// TIA Portal project "MobileLLRF" (V18)

(* hardware
DEVICE "S7-1200 station_1"  S7-1200 Station
   slot 0: "Rack_0"  S7-1200 Rack  Rack  V1.0
   slot 1: "PLC_1"  CPU 1212C DC/DC/DC  6ES7 212-1AE40-0XB0  V4.6
   slot 3: "AQ 1x12BIT_1"  AQ1 signal board  6ES7 232-4HA30-0XB0  V1.0
*)

// ===== PLC "PLC_1"  CPU 1212C DC/DC/DC =====

VAR_GLOBAL   // PLC tag table "Default tag table"
   "System_Byte" AT %MB1 : Byte;
   "FirstScan" AT %M1.0 : Bool;
   "DiagStatusUpdate" AT %M1.1 : Bool;
   "AlwaysTRUE" AT %M1.2 : Bool;
   "AlwaysFALSE" AT %M1.3 : Bool;
   "Clock_Byte" AT %MB0 : Byte;
   "Clock_10Hz" AT %M0.0 : Bool;
   "Clock_5Hz" AT %M0.1 : Bool;
   "Clock_2.5Hz" AT %M0.2 : Bool;
   "Clock_2Hz" AT %M0.3 : Bool;
   "Clock_1.25Hz" AT %M0.4 : Bool;
   "Clock_1Hz" AT %M0.5 : Bool;
   "Clock_0.625Hz" AT %M0.6 : Bool;
   "Clock_0.5Hz" AT %M0.7 : Bool;
END_VAR

VAR_GLOBAL   // PLC tag table "In/Out"
   "DigitalInputs" AT %IB0 : Byte;
   "DigitalOutputs" AT %QB0 : Byte;
   "AI0" AT %IW64 : Int;
   "AI1" AT %IW66 : Int;
   "TestDO" AT %Q0.5 : Bool;
   "AQ0" AT %QW80 : Int;
   "AI_Combined" AT %ID64 : DWord;
   "TriggerLED" AT %Q0.0 : Bool;
END_VAR

TYPE "PLC2Epics_TYPE"
   STRUCT
      CavPos0 : Bool;
      CavPos1 : Bool;
      CavPos2 : Bool;
      RFswitchON : Bool;
      StepAtten10dB : Bool;
      StepAtten20dB : Bool;
      StepAtten40dB : Bool;
      SSPAenabled : Bool;
      ExtIntrlk : Bool;
      VCA_Ctrl : Real;
      spare : Array[0..9] of Word;
   END_STRUCT;
END_TYPE

TYPE "Epics2PLC_TYPE"
   STRUCT
      StepAtten10dB : Bool;
      StepAtten20dB : Bool;
      StepAtten40dB : Bool;
      RFswitchON : Bool;
      EnableSSPA : Bool;
      VCA_Ctrl : Real;
      spare : Array[0..9] of Word;
   END_STRUCT;
END_TYPE

TYPE "CommParam"
VERSION : 0.1
   STRUCT
      interface_id : Word;   // HW-identifier of IE-interface submodule
      conn_id : Word;   // Connection reference / identifier
      connection_type : Byte := 16#000B;   // Type of connection: 11=TCP/IP, 19=UDP (17=TCP/IP) ??B#16#11??
      active_established : Bool := False;   // active/passive connection establishment
      local_port : UInt;   // local UDP/TCP port number
      init_com : Bool;   // send_db : INT; recv_db : INT;
      send_len : UDInt;
      recv_len : UDInt;
      sendtrigger : Bool;
      sendtime : Time_Of_Day;
      sendinterval : DInt;
   END_STRUCT;
END_TYPE

// folder: EPICS_Communication

DATA_BLOCK "CH_PARAM_TCP"   // DB300
{ S7_Optimized_Access := 'FALSE' }
VERSION : 0.1
   VAR
      CommParam : "CommParam";
   END_VAR
BEGIN
   CommParam.send_len := 26;
   CommParam.recv_len := 26;
   CommParam.sendinterval := DINT#500;
   CommParam.local_port := 3000;
   CommParam.interface_id := 64;
   CommParam.conn_id := 3;
   CommParam.connection_type := 16#000b;
END_DATA_BLOCK

DATA_BLOCK "TCP1_instance"   // DB310
{ S7_Optimized_Access := 'FALSE' }
AUTHOR : CSL
FAMILY : TSTMP
NAME : S_R_TCP1
VERSION : 1.0
// stored: InstanceOfName Tsend_Trecv
"Tsend_Trecv"
BEGIN
END_DATA_BLOCK

// folder: Epics

DATA_BLOCK "PLC2Epics"   // DB100
{ S7_Optimized_Access := 'FALSE' }
VERSION : 0.1
   VAR
      DATA : "PLC2Epics_TYPE";
   END_VAR
BEGIN
END_DATA_BLOCK

DATA_BLOCK "Epics2PLC"   // DB101
{ S7_Optimized_Access := 'FALSE' }
VERSION : 0.1
   VAR
      data : "Epics2PLC_TYPE";
   END_VAR
BEGIN
END_DATA_BLOCK

// folder: Input/Output

DATA_BLOCK "#ANALOG_IN"   // DB400
{ S7_Optimized_Access := 'FALSE' }
VERSION : 0.1
   VAR
      Spare1 : Int;
      Spare2 : Int;
   END_VAR
BEGIN
END_DATA_BLOCK

DATA_BLOCK "#ANALOG_OUT"   // DB401
{ S7_Optimized_Access := 'FALSE' }
VERSION : 0.1
   VAR
      VCA_Ctrl : Word;
   END_VAR
BEGIN
END_DATA_BLOCK

DATA_BLOCK "#DIGITAL_INPUTS"   // DB402
{ S7_Optimized_Access := 'FALSE' }
VERSION : 0.1
   VAR
      CavPos0 : Bool;   // Coded LLRF connection to DUT (LSB)
      CavPos1 : Bool;   // Coded LLRF connection to DUT
      CavPos2 : Bool;   // Coded LLRF connection to DUT (MSB)
      RFswitchOn : Bool;
      ExtIntlk : Bool;
      Spare2 : Bool;
      Spare3 : Bool;
      Spare4 : Bool;
   END_VAR
BEGIN
END_DATA_BLOCK

DATA_BLOCK "#DIGITAL_OUTPUTS"   // DB403
{ S7_Optimized_Access := 'FALSE' }
VERSION : 0.1
   VAR
      StepAtt10dB : Bool;
      StepAtt20dB : Bool;
      StepAtt40dB : Bool;
      RFswitchOff : Bool;
      RFswitchOn : Bool;
      EnableSSPA : Bool;
   END_VAR
BEGIN
END_DATA_BLOCK

// folder: (top level)

FUNCTION "Process" : Void   // FC103, LAD
TITLE = Process logic
{ S7_Optimized_Access := 'TRUE' }
VERSION : 0.1
BEGIN

REGION Network 1
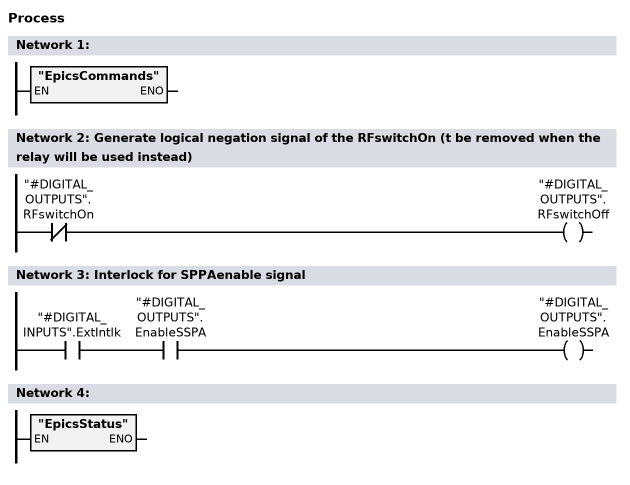
   RUNG wire#powerrail
      "EpicsCommands"()
   END_RUNG
   // the same network as SCL:
   "EpicsCommands"();
END_REGION

REGION Network 2: Generate logical negation signal of the RFswitchOn (t be removed when the relay will be used instead)
   RUNG wire#powerrail
      I_Contact( "#DIGITAL_OUTPUTS".RFswitchOn )
      Coil( "#DIGITAL_OUTPUTS".RFswitchOff )
   END_RUNG
   // the same network as SCL:
   "#DIGITAL_OUTPUTS".RFswitchOff := NOT "#DIGITAL_OUTPUTS".RFswitchOn;
END_REGION

REGION Network 3: Interlock for SPPAenable signal
   RUNG wire#powerrail
      Contact( "#DIGITAL_INPUTS".ExtIntlk )
      Contact( "#DIGITAL_OUTPUTS".EnableSSPA )
      Coil( "#DIGITAL_OUTPUTS".EnableSSPA )
   END_RUNG
   // the same network as SCL:
   "#DIGITAL_OUTPUTS".EnableSSPA := "#DIGITAL_INPUTS".ExtIntlk AND "#DIGITAL_OUTPUTS".EnableSSPA;
END_REGION

REGION Network 4
   RUNG wire#powerrail
      "EpicsStatus"()
   END_RUNG
   // the same network as SCL:
   "EpicsStatus"();
END_REGION
END_FUNCTION

ORGANIZATION_BLOCK "Main"   // OB1, LAD, ProgramCycle
TITLE = "Main Program Sweep (Cycle)"
{ S7_Optimized_Access := 'TRUE' }
VERSION : 0.1
   VAR_INPUT
      Initial_Call : Bool;   // Initial call of this OB
      Remanence : Bool;   // =True, if remanent data are available
   END_VAR
BEGIN

REGION Network 1
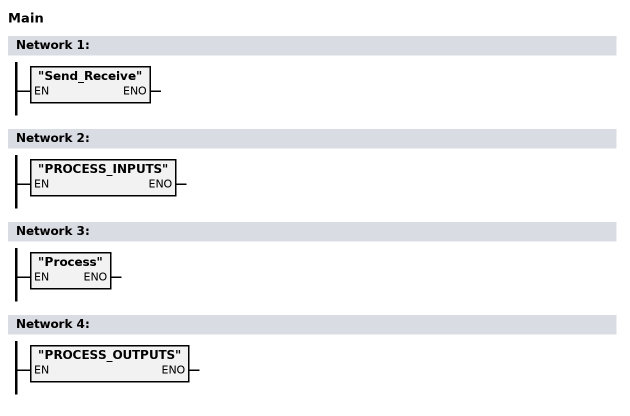
   RUNG wire#powerrail
      "Send_Receive"()
   END_RUNG
   // the same network as SCL:
   "Send_Receive"();
END_REGION

REGION Network 2
   RUNG wire#powerrail
      "PROCESS_INPUTS"()
   END_RUNG
   // the same network as SCL:
   "PROCESS_INPUTS"();
END_REGION

REGION Network 3
   RUNG wire#powerrail
      "Process"()
   END_RUNG
   // the same network as SCL:
   "Process"();
END_REGION

REGION Network 4
   RUNG wire#powerrail
      "PROCESS_OUTPUTS"()
   END_RUNG
   // the same network as SCL:
   "PROCESS_OUTPUTS"();
END_REGION
END_ORGANIZATION_BLOCK

ORGANIZATION_BLOCK "Startup"   // OB100, LAD, Startup
TITLE = "Complete Restart"
{ S7_Optimized_Access := 'TRUE' }
VERSION : 0.1
   VAR_INPUT
      LostRetentive : Bool;   // True if retentive data are lost
      LostRTC : Bool;   // True if date and time are lost
   END_VAR
BEGIN

REGION Network 1
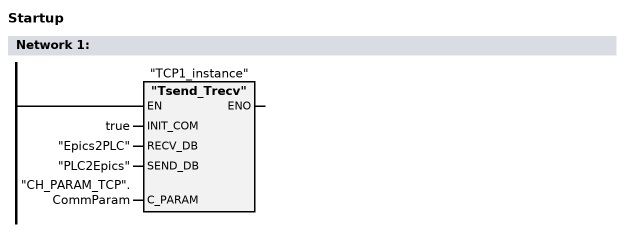
   RUNG wire#powerrail
      "TCP1_instance"(INIT_COM := true, RECV_DB := "Epics2PLC", SEND_DB := "PLC2Epics", C_PARAM := "CH_PARAM_TCP".CommParam)
   END_RUNG
   // the same network as SCL:
   "TCP1_instance"(INIT_COM := true,   // "Tsend_Trecv"
                   RECV_DB := "Epics2PLC",
                   SEND_DB := "PLC2Epics",
                   C_PARAM := "CH_PARAM_TCP".CommParam);
END_REGION
END_ORGANIZATION_BLOCK

// folder: EPICS_Communication

FUNCTION_BLOCK "Tsend_Trecv"   // FB300, SCL
TITLE = TCP1 send receive channel
{ S7_Optimized_Access := 'FALSE' }
AUTHOR : CSL
FAMILY : TSTMP
NAME : S_R_TCP1
VERSION : 1.0
   VAR_INPUT
      INIT_COM : Bool;
      RECV_DB : Variant;
      SEND_DB : Variant;
   END_VAR
   VAR_IN_OUT
      C_PARAM : "CommParam";
   END_VAR
   VAR
      T_SEND : TSEND;
      T_RECV : TRCV;
      T_CONN : TCON;
      T_PARAM : TCON_IP_v4;
      COM1 : Struct
         CONNECTED : Bool;
         CONN_DONE : Bool;
         CONN_BUSY : Bool;
         CONN_ERROR : Bool;
         CONN_STATUS : Word;
         CONN_SETA : Bool;
         SEND_REQ : Bool;
         SEND_DONE : Bool;
         SEND_BUSY : Bool;
         SEND_ERROR : Bool;
         SEND_REQ_P : Bool;
         SEND_STATUS : Word;
         ACT_SEND : Bool;
         RECV_NDR : Bool;
         RECV_BUSY : Bool;
         RECV_ERROR : Bool;
         RECV_STATUS : Word;
         RECV_LEN : UDInt;
      END_STRUCT;
      PLC_COUNT : UDInt;
      CURRENT_DT : DTL;
   END_VAR
   VAR_TEMP
      current_time : Time;
      TIME_DIFF : DInt;
      SEND_TIME : DInt;
      stat : Int;
      tod : Time_Of_Day;
   END_VAR
   VAR CONSTANT
      DAY_IN_MS : DInt := 86400000;
   END_VAR
BEGIN

   // Set communication initialisation bit at restart
   #C_PARAM.init_com := #INIT_COM;

   //Clear Bits to start initial connection and communication
   IF #C_PARAM.init_com THEN
       #COM1.CONNECTED := FALSE;
       #COM1.SEND_REQ := FALSE;
       #COM1.CONN_SETA := FALSE;
   END_IF;

   //set TCPx connection parametres 
   #T_PARAM.InterfaceId :=  WORD_TO_UINT (#C_PARAM.interface_id);
   #T_PARAM.ID := #C_PARAM.conn_id;
   #T_PARAM.ConnectionType := #C_PARAM.connection_type;
   #T_PARAM.ActiveEstablished := #C_PARAM.active_established;
   //T_PARAM.RemotePort := 0; 
   #T_PARAM.LocalPort := #C_PARAM.local_port;

   //Establish TCP connection
   //After the connection has been established, it is automatically monitored and maintained by the operating system of the CPU.
   //If the connection has been interrupted, by any line break or due to the remote communications partner, the active partner attempts to reestablish the connection.
   //Therefore, the FB 65 "TCON" may not be called again! 
   IF NOT #COM1.CONNECTED THEN
       #T_CONN(REQ := #COM1.CONN_SETA,
               ID := #C_PARAM.conn_id,
               DONE => #COM1.CONN_DONE,
               BUSY => #COM1.CONN_BUSY,
               ERROR => #COM1.CONN_ERROR,
               STATUS => #COM1.CONN_STATUS,
               CONNECT := #T_PARAM);
   END_IF;

   //Establish connection
   //While startup phase (initial).
   //Indication of the connection status:
   //a) If the CPU may establish the specified connection after Stop/Run immediately, the variable "CONNECTED" indicates HIGH (=1).
   //b) If the CPU is not able to establish the specified connection after Stop/Run, the variable "CONNECTED" remains LOW(=0).
   //c) Note: If the instance DB is loaded by the user, the variable "CONNECTED" indicates HIGH, although the connection may not be established yet. 
   //However, the FB64 "TRCV" would indicate the STATUS=0x80C4, as long as the connection has NOT been established. 
   IF #C_PARAM.init_com THEN
       #COM1.CONN_SETA := TRUE;
   END_IF;
   IF #COM1.CONN_DONE THEN
       #COM1.CONN_SETA := FALSE;
       #C_PARAM.init_com := FALSE;
   END_IF;
   IF #COM1.CONN_SETA THEN
       #COM1.CONNECTED := FALSE;
   ELSE
       #COM1.CONNECTED := TRUE;
   END_IF;

   //generate send trigger pulse
   //#current_time := TIME_TCK(); // Not available in S/-1200 
   #stat := RD_SYS_T(#CURRENT_DT); // TIME & DATE
   #tod := DTL_TO_TOD(#CURRENT_DT); // Time of Day (ms after midnight)
   #TIME_DIFF := TOD_TO_DINT(#tod) - TOD_TO_DINT(#C_PARAM.sendtime);
   IF (#TIME_DIFF < 0) THEN
       #TIME_DIFF := #TIME_DIFF + #DAY_IN_MS;
   END_IF;
   IF (#C_PARAM.sendinterval < #TIME_DIFF + 1) THEN
       #C_PARAM.sendtrigger := TRUE;
       #SEND_TIME := TOD_TO_DINT(#C_PARAM.sendtime) + #C_PARAM.sendinterval;
       IF (#SEND_TIME >= #DAY_IN_MS) THEN
           #SEND_TIME := #SEND_TIME - #DAY_IN_MS;
       END_IF;
       #C_PARAM.sendtime := DINT_TO_TOD(#SEND_TIME);
       #COM1.SEND_REQ_P := FALSE;
   END_IF;
   //IF (#C_PARAM.sendinterval < ABS(TIME_TO_DINT(#current_time - #C_PARAM.sendtime)) + 1) THEN
   //    #C_PARAM.sendtrigger := TRUE;
   //    #C_PARAM.sendtime := #C_PARAM.sendtime + DINT_TO_TIME(#C_PARAM.sendinterval);  //#C_PARAM.sendtime := #current_time;
   //    #COM1.SEND_REQ_P := FALSE;
   // END_IF;

   //Invoke T_SEND function. 
   //IF connection is established TO transmit the data TO the partner as a message.
   // DATA and LEN from input C_PARAM
   IF #COM1.CONNECTED THEN
       #T_SEND(REQ := #COM1.SEND_REQ,
               ID := #C_PARAM.conn_id,
               LEN := #C_PARAM.send_len,
               DONE => #COM1.SEND_DONE,
               BUSY => #COM1.SEND_BUSY,
               ERROR => #COM1.SEND_ERROR,
               STATUS => #COM1.SEND_STATUS,
               DATA := #SEND_DB);//"datatoIOC_TCP1".CommToIOC);
   END_IF;

   //Generate the rising edge SEND_REQ to start the T_SEND function. 
   IF #C_PARAM.sendtrigger AND NOT #COM1.SEND_REQ_P AND NOT #COM1.SEND_BUSY THEN
        #COM1.SEND_REQ := TRUE;
   END_IF;
   #COM1.SEND_REQ_P := #C_PARAM.sendtrigger;

   IF #COM1.SEND_DONE OR #COM1.SEND_ERROR THEN
       #COM1.SEND_REQ := FALSE;
       #C_PARAM.sendtrigger := FALSE;
   END_IF;


   //Invoke T_RECV function
   //The data is stored into the buffer specified with DATA parameter. 
   //After the data has been received, the data is immediately available in the receive buffer. 
   //Receiving is indicated BY the NDR output parameter.
   //Note: DATA and LEN from input C_PARAM 
   IF #COM1.CONNECTED THEN
       #T_RECV(EN_R := #COM1.CONNECTED,
               ID := #C_PARAM.conn_id,
               LEN := #C_PARAM.recv_len,
               ADHOC := false,
               NDR => #COM1.RECV_NDR,
               BUSY => #COM1.RECV_BUSY,
               ERROR => #COM1.RECV_ERROR,
               STATUS => #COM1.RECV_STATUS,
               RCVD_LEN => #COM1.RECV_LEN,
               DATA := #RECV_DB);//"datatoPLC_TCP1".CommToPLC);  

       //Send by request
       //IF (#T_RECV.RCVD_LEN > 0) THEN
       //    #COM1.SEND_REQ := TRUE;
       //END_IF;

   END_IF;
END_FUNCTION_BLOCK

FUNCTION "Send_Receive" : Void   // FC105, SCL
TITLE = Send and receive
{ S7_Optimized_Access := 'FALSE' }
AUTHOR : CSL
FAMILY : TSTMP
NAME : snd_rcv
VERSION : 1.0
BEGIN
   // "channel_param_TCP1".cParam.enable := true;
   //"CH_PARAM_TCP".TCP2_Instance.cParam.enable := true;
   //"CH_PARAM_TCP".TCP3_Instance.cParam.enable := true;
   //

   // Initialize the connection (open the port for listening)
   // 
   // Uncomment the IF block below or call "TCP1_instance"(INIT_COM := TRUE,...) in Startup block (OB100)
   // 
   //IF ("FirstScan") THEN
   //    "TCP1_instance"(INIT_COM := TRUE,
   //                    RECV_DB := "Epics2PLC",
   //                    SEND_DB := "PLC2Epics",
   //                    C_PARAM := "CH_PARAM_TCP_CPU".CommParam);     // IN_OUT: STRUCT
   //END_IF;

   "TCP1_instance"(INIT_COM := False,
                   RECV_DB := "Epics2PLC",
                   SEND_DB := "PLC2Epics",
                   C_PARAM := "CH_PARAM_TCP".CommParam);     // IN_OUT: STRUCT
END_FUNCTION

// folder: Epics

FUNCTION "EpicsStatus" : Void   // FC100, LAD
{ S7_Optimized_Access := 'TRUE' }
VERSION : 0.1
// Send data to Epics
   VAR_TEMP
      tmp : Real;
   END_VAR
BEGIN

REGION Network 1: CavPos0
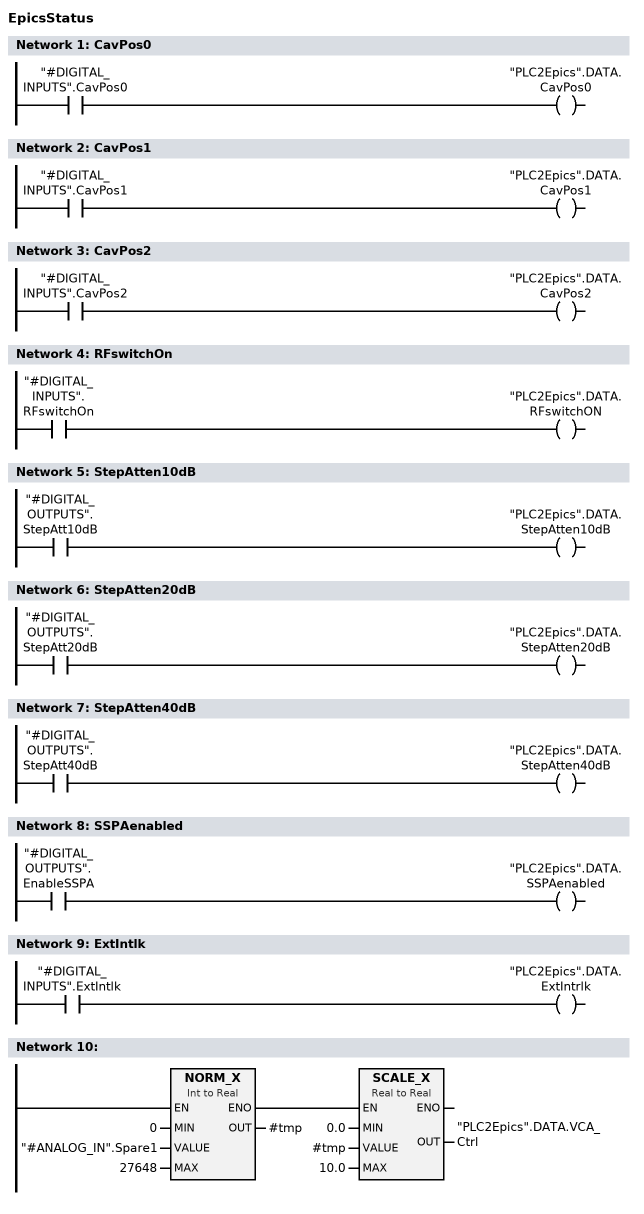
   RUNG wire#powerrail
      Contact( "#DIGITAL_INPUTS".CavPos0 )
      Coil( "PLC2Epics".DATA.CavPos0 )
   END_RUNG
   // the same network as SCL:
   "PLC2Epics".DATA.CavPos0 := "#DIGITAL_INPUTS".CavPos0;
END_REGION

REGION Network 2: CavPos1
   RUNG wire#powerrail
      Contact( "#DIGITAL_INPUTS".CavPos1 )
      Coil( "PLC2Epics".DATA.CavPos1 )
   END_RUNG
   // the same network as SCL:
   "PLC2Epics".DATA.CavPos1 := "#DIGITAL_INPUTS".CavPos1;
END_REGION

REGION Network 3: CavPos2
   RUNG wire#powerrail
      Contact( "#DIGITAL_INPUTS".CavPos2 )
      Coil( "PLC2Epics".DATA.CavPos2 )
   END_RUNG
   // the same network as SCL:
   "PLC2Epics".DATA.CavPos2 := "#DIGITAL_INPUTS".CavPos2;
END_REGION

REGION Network 4: RFswitchOn
   RUNG wire#powerrail
      Contact( "#DIGITAL_INPUTS".RFswitchOn )
      Coil( "PLC2Epics".DATA.RFswitchON )
   END_RUNG
   // the same network as SCL:
   "PLC2Epics".DATA.RFswitchON := "#DIGITAL_INPUTS".RFswitchOn;
END_REGION

REGION Network 5: StepAtten10dB
   RUNG wire#powerrail
      Contact( "#DIGITAL_OUTPUTS".StepAtt10dB )
      Coil( "PLC2Epics".DATA.StepAtten10dB )
   END_RUNG
   // the same network as SCL:
   "PLC2Epics".DATA.StepAtten10dB := "#DIGITAL_OUTPUTS".StepAtt10dB;
END_REGION

REGION Network 6: StepAtten20dB
   RUNG wire#powerrail
      Contact( "#DIGITAL_OUTPUTS".StepAtt20dB )
      Coil( "PLC2Epics".DATA.StepAtten20dB )
   END_RUNG
   // the same network as SCL:
   "PLC2Epics".DATA.StepAtten20dB := "#DIGITAL_OUTPUTS".StepAtt20dB;
END_REGION

REGION Network 7: StepAtten40dB
   RUNG wire#powerrail
      Contact( "#DIGITAL_OUTPUTS".StepAtt40dB )
      Coil( "PLC2Epics".DATA.StepAtten40dB )
   END_RUNG
   // the same network as SCL:
   "PLC2Epics".DATA.StepAtten40dB := "#DIGITAL_OUTPUTS".StepAtt40dB;
END_REGION

REGION Network 8: SSPAenabled
   RUNG wire#powerrail
      Contact( "#DIGITAL_OUTPUTS".EnableSSPA )
      Coil( "PLC2Epics".DATA.SSPAenabled )
   END_RUNG
   // the same network as SCL:
   "PLC2Epics".DATA.SSPAenabled := "#DIGITAL_OUTPUTS".EnableSSPA;
END_REGION

REGION Network 9: ExtIntlk
   RUNG wire#powerrail
      Contact( "#DIGITAL_INPUTS".ExtIntlk )
      Coil( "PLC2Epics".DATA.ExtIntrlk )
   END_RUNG
   // the same network as SCL:
   "PLC2Epics".DATA.ExtIntrlk := "#DIGITAL_INPUTS".ExtIntlk;
END_REGION

REGION Network 10
   RUNG wire#powerrail
      { S7_Templates := "[SrcType := Int, DestType := Real]" } Normalize(min := 0, value := "#ANALOG_IN".Spare1, max := 27648, out => #tmp)
      { S7_Templates := "[SrcType := Real, DestType := Real]" } Scale(min := 0.0, value := #tmp, max := 10.0, out => "PLC2Epics".DATA.VCA_Ctrl)
   END_RUNG
   // the same network as SCL:
   #tmp := NORM_X(MIN := 0, VALUE := "#ANALOG_IN".Spare1, MAX := 27648);
   "PLC2Epics".DATA.VCA_Ctrl := SCALE_X(MIN := 0.0, VALUE := #tmp, MAX := 10.0);
END_REGION
END_FUNCTION

FUNCTION "EpicsCommands" : Void   // FC101, LAD
{ S7_Optimized_Access := 'TRUE' }
VERSION : 0.1
// Get data from Epics
   VAR_TEMP
      tmp : Real;
   END_VAR
BEGIN

REGION Network 1: StepAtten10dB
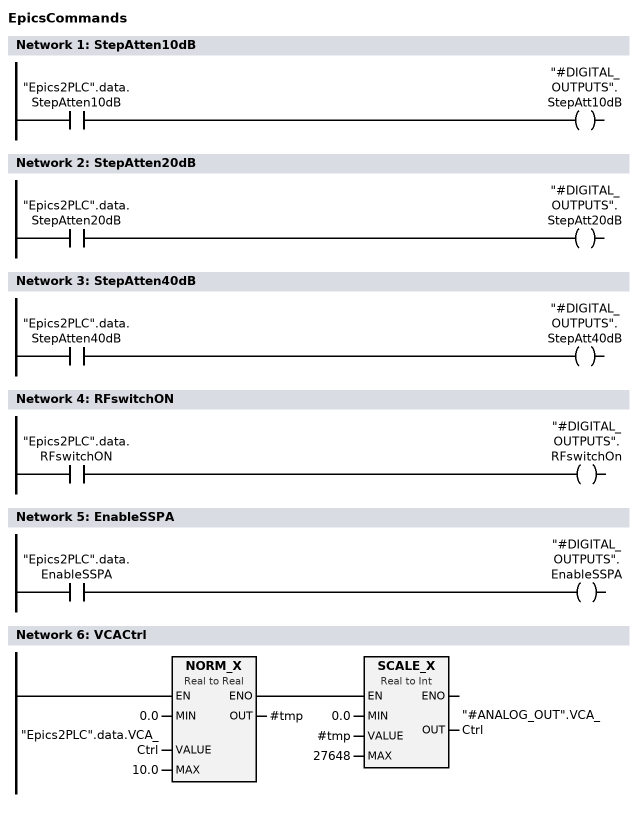
   RUNG wire#powerrail
      Contact( "Epics2PLC".data.StepAtten10dB )
      Coil( "#DIGITAL_OUTPUTS".StepAtt10dB )
   END_RUNG
   // the same network as SCL:
   "#DIGITAL_OUTPUTS".StepAtt10dB := "Epics2PLC".data.StepAtten10dB;
END_REGION

REGION Network 2: StepAtten20dB
   RUNG wire#powerrail
      Contact( "Epics2PLC".data.StepAtten20dB )
      Coil( "#DIGITAL_OUTPUTS".StepAtt20dB )
   END_RUNG
   // the same network as SCL:
   "#DIGITAL_OUTPUTS".StepAtt20dB := "Epics2PLC".data.StepAtten20dB;
END_REGION

REGION Network 3: StepAtten40dB
   RUNG wire#powerrail
      Contact( "Epics2PLC".data.StepAtten40dB )
      Coil( "#DIGITAL_OUTPUTS".StepAtt40dB )
   END_RUNG
   // the same network as SCL:
   "#DIGITAL_OUTPUTS".StepAtt40dB := "Epics2PLC".data.StepAtten40dB;
END_REGION

REGION Network 4: RFswitchON
   RUNG wire#powerrail
      Contact( "Epics2PLC".data.RFswitchON )
      Coil( "#DIGITAL_OUTPUTS".RFswitchOn )
   END_RUNG
   // the same network as SCL:
   "#DIGITAL_OUTPUTS".RFswitchOn := "Epics2PLC".data.RFswitchON;
END_REGION

REGION Network 5: EnableSSPA
   RUNG wire#powerrail
      Contact( "Epics2PLC".data.EnableSSPA )
      Coil( "#DIGITAL_OUTPUTS".EnableSSPA )
   END_RUNG
   // the same network as SCL:
   "#DIGITAL_OUTPUTS".EnableSSPA := "Epics2PLC".data.EnableSSPA;
END_REGION

REGION Network 6: VCACtrl
   RUNG wire#powerrail
      { S7_Templates := "[SrcType := Real, DestType := Real]" } Normalize(min := 0.0, value := "Epics2PLC".data.VCA_Ctrl, max := 10.0, out => #tmp)
      { S7_Templates := "[SrcType := Real, DestType := Int]" } Scale(min := 0.0, value := #tmp, max := 27648, out => "#ANALOG_OUT".VCA_Ctrl)
   END_RUNG
   // the same network as SCL:
   #tmp := NORM_X(MIN := 0.0, VALUE := "Epics2PLC".data.VCA_Ctrl, MAX := 10.0);
   "#ANALOG_OUT".VCA_Ctrl := SCALE_X(MIN := 0.0, VALUE := #tmp, MAX := 27648);
END_REGION
END_FUNCTION

// folder: Input/Output

FUNCTION "PROCESS_INPUTS" : Void   // FC400, LAD
{ S7_Optimized_Access := 'TRUE' }
VERSION : 0.1
   VAR_TEMP
      status : Word;
   END_VAR
BEGIN

REGION Network 1: Read digital inputs (8)
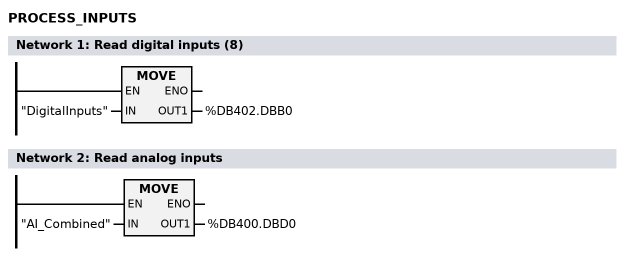
   RUNG wire#powerrail
      Move(in := "DigitalInputs", out1 => %DB402.DBB0)
   END_RUNG
   // the same network as SCL:
   %DB402.DBB0 := "DigitalInputs";
END_REGION

REGION Network 2: Read analog inputs
   RUNG wire#powerrail
      Move(in := "AI_Combined", out1 => %DB400.DBD0)
   END_RUNG
   // the same network as SCL:
   %DB400.DBD0 := "AI_Combined";
END_REGION
END_FUNCTION

FUNCTION "PROCESS_OUTPUTS" : Void   // FC401, LAD
{ S7_Optimized_Access := 'TRUE' }
VERSION : 0.1
   VAR_TEMP
      status : Word;
   END_VAR
BEGIN

REGION Network 1: Write digital outputs (6)
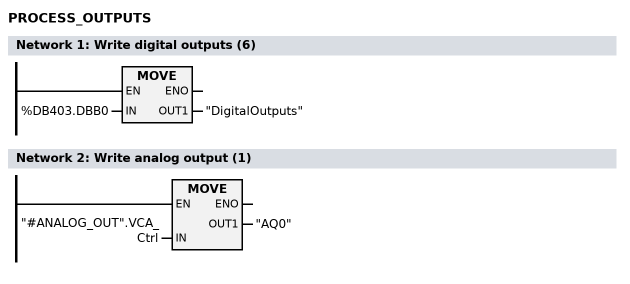
   RUNG wire#powerrail
      Move(in := %DB403.DBB0, out1 => "DigitalOutputs")
   END_RUNG
   // the same network as SCL:
   "DigitalOutputs" := %DB403.DBB0;
END_REGION

REGION Network 2: Write analog output (1)
   RUNG wire#powerrail
      Move(in := "#ANALOG_OUT".VCA_Ctrl, out1 => "AQ0")
   END_RUNG
   // the same network as SCL:
   "AQ0" := "#ANALOG_OUT".VCA_Ctrl;
END_REGION
END_FUNCTION

// ===== library types =====

TYPE "CPU_WCONF"
VERSION : 0.0
   STRUCT
      RESET : Bool;   // CPU reset command
      OFF : Bool;   // OFF Command
      EE_1_CLOSE : Bool;   // Auxiliary Command
      EE_1_RESET : Bool;   // Filament Command
      EE_2_CLOSE : Bool;   // Standby command
      EE_2_RESET : Bool;   // High-voltage ON command
      RFON : Bool;   // RF ON command
      TEST_ALL_AD : Bool;   // Test all arc detectors
      WR_DATA : Bool;   // Write data into the read DB
      OP_MODE : Byte;   // 1 = Bypass mode, 2 = Maintenance/testing mode, 3 = Normal operation, 4 = Wire test
   END_STRUCT;
END_TYPE

TYPE "CPU_RCONF"
VERSION : 0.0
   STRUCT
      RESET : Bool;   // CPU reset command
      LATCH_MODE : Bool;   // CPU latching mode
      INTERLOCK : Bool;   // CPU Interlock/Alarm
      ACK_REQ : Bool;   // CPU Warning
      GERSEMI_COM_OK : Bool;   // Communication with Gersemi OK
      FLSHBX_HV : Bool;   // Flash Box High Voltage
      FLSHBX_HC : Bool;   // Flash Box High Current
      FLSHBX_He : Bool;   // Flash Box Helium
      RFON_MISS_COND : Bool;   // RF Enable missed condition
      AUX_SUP_COND : Bool;   // AUX missed supervision
      FIL_SUP_COND : Bool;   // FIL missed supervision
      STDBY_SUP_COND : Bool;   // STDBY missed supervision
      HVON_SUP_COND : Bool;   // HVON missed supervision
      RFON_SUP_COND : Bool;   // RFON missed supervision
      OFF : Bool;   // OFF Command
      EE_1_CLOSE : Bool;   // Auxiliary Command
      EE_1_RESET : Bool;   // Filament Command
      EE_2_CLOSE : Bool;   // Standby command
      EE_2_RESET : Bool;   // High-voltage ON command
      RFON : Bool;   // RF ON command
      FORCE_DIS_MODE_ACT : Bool;   // One or more signals are being disabled or forced
      TEST_ALL_AD : Bool;   // Test all arc detectors
      ACT_STAT : Byte;   // Actual State
      SET_STATE : Int;   // Set State to the target
      OP_MODE : Byte;   // 1 = Bypass mode, 2 = Maintenance/testing mode, 3 = Normal operation, 4 = Wire test
   END_STRUCT;
END_TYPE